(*

.. <legal notes>

legal notes
=================
| SPDX-FileCopyrightText: © 2025 Oleksandr Tiutyk <trofimich@gmail.com>
| SPDX-License-Identifier: LGPL-3.0-only
| For details check: LGPL-3.0-only_

.. _LGPL-3.0-only: https://www.gnu.org/licenses/lgpl-3.0.en.html

.. </legal notes>

*)

{attribute 'qualified_only'}
{attribute 'strict'}
{attribute 'to_string'}
TYPE AUTOMATION_CONTROLLER_STATE :
(
	INITIALIZING := 0,
    RUNNING := 1,            
    STOPPING := 2,            
    FAULT := 4 // Any error occurred while initializing or fatal error in other state
);
END_TYPE

(* stored: Version 1.1.0.1
   DUT AUTOMATION_CONTROLLER_STATE: Id {dc71eb7c-dbf6-4e3e-9f47-6ac56d62b3ac} *)
